(* PLC project  *)

PROGRAM P
  VAR  (* added by the conversion: wires and edge detectors of the diagram *)
    _AND3_OUT : BOOL;
  END_VAR

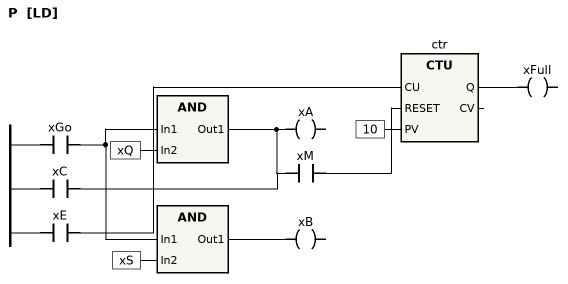
(* LD diagram, written out as Structured Text *)
_AND3_OUT := xGo AND xQ;
xA := _AND3_OUT;
xB := xGo AND xS;
ctr(CU := xE, RESET := (_AND3_OUT OR xC) AND xM, PV := 10);
xFull := ctr.Q;
END_PROGRAM
